FUNCTION_BLOCK Composite
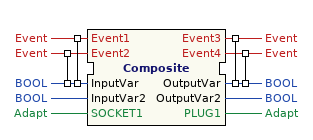
  EVENT_INPUT
    Event1 WITH InputVar;
    Event2 WITH InputVar;
  END_EVENT
  EVENT_OUTPUT
    Event3 WITH OutputVar;
    Event4 WITH OutputVar;
  END_EVENT
  VAR_INPUT
    InputVar : BOOL;
    InputVar2 : BOOL;
  END_VAR
  VAR_OUTPUT
    OutputVar : BOOL;
    OutputVar2 : BOOL;
  END_VAR
  SOCKETS
    SOCKET1 : Adapt;
  END_SOCKETS
  PLUGS
    PLUG1 : Adapt;
  END_PLUGS
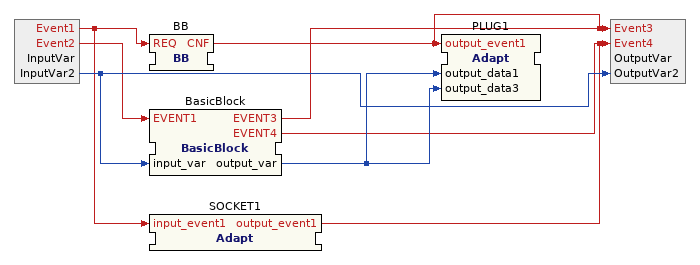
  FBS
    BB : BB;
    BasicBlock : BasicBlock;
  END_FBS
  EVENT_CONNECTIONS
    Event1 TO SOCKET1.input_event1;
    SOCKET1.output_event1 TO Event4;
    BasicBlock.EVENT3 TO Event3;
    BasicBlock.EVENT4 TO Event4;
    Event2 TO BasicBlock.EVENT1;
    BB.CNF TO Event3;
    Event1 TO BB.REQ;
    BB.CNF TO PLUG1.output_event1;
  END_CONNECTIONS
  DATA_CONNECTIONS
    InputVar2 TO BasicBlock.input_var;
    InputVar2 TO OutputVar2;
    BasicBlock.output_var TO PLUG1.output_data1;
    BasicBlock.output_var TO PLUG1.output_data3;
  END_CONNECTIONS
END_FUNCTION_BLOCK
